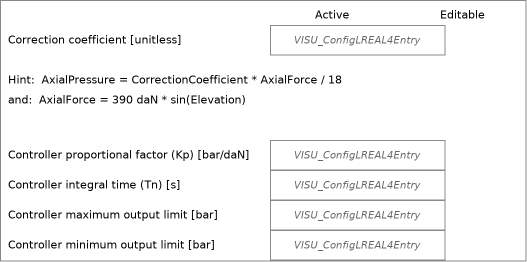
VISUALIZATION VISU_M1Config_Axial_General  // 527x262
VAR_IN_OUT
    editable : M1AxialSupportConfig;
	active : M1AxialSupportConfig;
END_VAR
    Label (270,5 125x20), "Active"
    Label (400,5 125x20), "Editable"
    Label (5,25 260x30), "Correction coefficient [unitless]"
    Frame (270,25 175x30)
        shows VISU_ConfigLREAL4Entry(active := active.correctionCoefficient, editable := editable.correctionCoefficient)
    Label (5,65 495x30), "Hint: AxialPressure = CorrectionCoefficient * AxialForce / 18"
    Label (5,85 495x30), "and: AxialForce = 390 daN * sin(Elevation)"
    Frame (270,140 175x30)
        shows VISU_ConfigLREAL4Entry(active := active.controllerKp, editable := editable.controllerKp)
    Label (5,140 260x30), "Controller proportional factor (Kp) [bar/daN]"
    Label (5,170 260x30), "Controller integral time (Tn) [s]"
    Frame (270,170 175x30)
        shows VISU_ConfigLREAL4Entry(active := active.controllerTn, editable := editable.controllerTn)
    Label (5,200 260x30), "Controller maximum output limit [bar]"
    Frame (270,200 175x30)
        shows VISU_ConfigLREAL4Entry(active := active.controllerLimitMax, editable := editable.controllerLimitMax)
    Frame (270,230 175x30)
        shows VISU_ConfigLREAL4Entry(active := active.controllerLimitMin, editable := editable.controllerLimitMin)
    Label (5,230 260x30), "Controller minimum output limit [bar]"
END_VISUALIZATION

(* stored: Version 1.1.0.1, ProductVersion 3.1.4019.2
   Visu VISU_M1Config_Axial_General: Id {e4e559fe-b98d-4217-ad1d-49688e95b15b} *)
